TYPE ST_BeamStabilizer :
STRUCT
	bError AT %I* : BOOL;
END_STRUCT
END_TYPE

(* stored: Version 1.1.0.1, ProductVersion 3.1.4022.17
   DUT ST_BeamStabilizer: Id {e4491502-131c-49e7-b3b3-d813ca570319} *)
